TYPE M3TranslationStatuses :
STRUCT
	healthStatus: HealthStatus;
	busyStatus: BusyStatus;
END_STRUCT
END_TYPE

(* stored: Version 1.1.0.1, ProductVersion 3.1.4019.2
   DUT M3TranslationStatuses: Id {7e145233-47db-4771-9113-db25c69bdc86} *)
